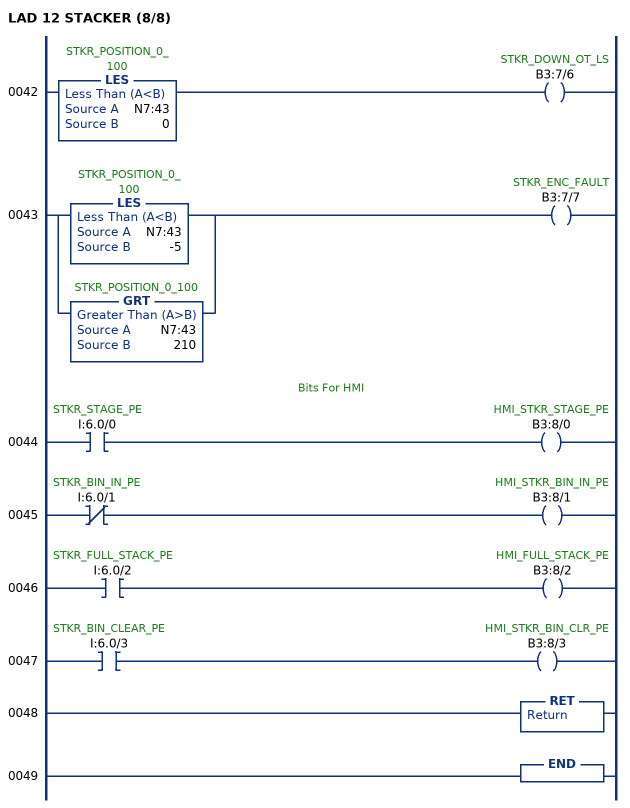
% Rung: 42 %
SOR LES N7:43 0 OTE B3:7/6 EOR
%   N7:43  STKR_POSITION_0_100 %
%   B3:7/6  STKR_DOWN_OT_LS %
% Rung: 43 %
SOR BST LES N7:43 -5 NXB GRT N7:43 210 BND OTE B3:7/7 EOR
%   N7:43  STKR_POSITION_0_100 %
%   B3:7/7  STKR_ENC_FAULT %
% Rung: 44 %
% Bits For HMI %
SOR XIC I:6.0/0 OTE B3:8/0 EOR
%   I:6.0/0  STKR_STAGE_PE %
%   B3:8/0  HMI_STKR_STAGE_PE %
% Rung: 45 %
SOR XIO I:6.0/1 OTE B3:8/1 EOR
%   I:6.0/1  STKR_BIN_IN_PE %
%   B3:8/1  HMI_STKR_BIN_IN_PE %
% Rung: 46 %
SOR XIC I:6.0/2 OTE B3:8/2 EOR
%   I:6.0/2  STKR_FULL_STACK_PE %
%   B3:8/2  HMI_FULL_STACK_PE %
% Rung: 47 %
SOR XIC I:6.0/3 OTE B3:8/3 EOR
%   I:6.0/3  STKR_BIN_CLEAR_PE %
%   B3:8/3  HMI_STKR_BIN_CLR_PE %
% Rung: 48 %
SOR RET EOR
% Rung: 49 %
SOR END EOR

OTHER DOCUMENTED ADDRESSES
  B3:0/9  SANITIZE_LTCH  "Triggered by reset limit sw."
  B3:0/10  SANITIZE_BIT  "Allow crdl ltch2 to unlatch only once until sanitize cycle is over"
  B3:0/11  CRDL_EN  "mcr on and no encoder fault"
  B3:0/15  CRDL_HAND_SS
  B3:1/1  RINSE_SELECT  "Turn ON Rinse"
  B3:1/9  RINSE_TEST
  B3:1/14  DUMP_INTERLOCK_SEL  "Dump Wash interlock"
  B3:2/7  UPPER_WASH_TEST
  B3:3/0  OPEN_CONTACT  "Machine not Equipt with OT LS"
  B3:3/9  FILTER_FLUSH_ON  "HMI Turn On Filter Flush"
  B3:3/11  MANUAL_BRUSH_DR_IN
  B3:3/12  MANUAL_BRUSH_DR_OUT
  B3:4/0  HMI_PID_MODE
  B3:4/1  HMI_PID_ALARM
  B3:6/11  BIN_STOP_DWN_SS
  C5:0/CU  EVENT_COUNTER
  F8:6  RAW_OUT_TO_VFD
  I:2.0/2  CHECK_MOTOR_OLS  "MP1,2,3,4,5"
  I:2.0/3  HP_PUMP_RUNNING
  I:2.0/4  CRADLE_VFD_RUNNING
  I:2.0/5  BRUSH_VFD_RUNNING
  I:2.0/6  XFER_PUMP_VFD_RUNNIN
  I:2.0/7  CRADLE_TORQUE_LIMIT
  I:5.0/3  BRUSH_GOING_IN
  I:5.0/4  BRUSH_GOING_OUT
  I:5.0/5  CRADLE_IN_MOTION
  I:5.0/6  BRUSH_RUNNING
  I:5.0/7  XFER_PUMP_RUNNING
  I:6.0  MAIN_TANK_RAW
  I:6.0/4  STKR_HI_LIMIT  "PROXIMITY SENSOR"
  L10:1/1  FAULT_MESSAGES
  N7:1/0  "Fault-Infeed Blocked"
  N7:1/1  "Fault-Outfeed Blocked"
  N7:1/2  "Fault-Cradle Overtravel Up"
  N7:1/3  "Fault-Cradle Overtravel down"
  N7:1/4  "Fault-Torque Cradle Inverter"
  N7:1/5  "Main Tank Low"
  N7:1/6  "Encoder Fault"
  N7:1/7  "Fill Main Tank"
  N7:10  FILTER_LOW_LS  "Filter Tank Low Level LS"
  N7:32  HP_PID_OUTPUT  "0-16383"
  N7:36  HMI_FLUSH_VALVE  "HMI TIME BETWEEN FLUSH"
  N7:37  HMI_FLUSH_VALVE_  "HMI FLUSHING TIME"
  N7:59  BIN_D_SLOW_DOWN
  N7:60  CATWALK_OPS_TIMER
  N9:0  K1
  O:0.0/7  CRADLE_COAST_TO_STOP  "MI2"
  O:0.0/12  FI
  O:0.1  OUT_TO_HP_VFD
  PD11:1  HIGH_PRESS_PUMP_PID
  PD11:1.2  PRESSURE_SP
  PD11:1.3  HP_KC
  PD11:1.4  HP_TI
  PD11:1.5  HP_TD
  PD11:1.13  LOOP_UPDATE_TIME  ".002"
  PD12:0.3  HP_PUMP_PID
  STKR_FULL_UP  
  T4:0/EN  CRDL_DWN_T  "Allows cradle to set down completely before conv starts"
  T4:1  CRDL_FLT_T1
  T4:2  CRDL_FLT_T2
  T4:5  CLEAN_CW_TMR  "CLOCKWISE CLEANING TIME"
  T4:6  SANITIZE_T
  T4:7  CRDL_DWN_T2  "Inhibits cradle up for 5 sec. after cradle sets down"
  T4:8  CLEAN_CCW  "COUNTER CLOCKWISE CLEANING TIME"
  T4:10  CRADLE_TIMER  "Cradle travel watch dog timer"
  T4:28/DN  LS_MED_BIN_DELAY
  T4:33/DN  STKR_RESTART_DELAY
  T4:34/DN  BIN_IN_DLY  "Stacker going down"
  T4:42  "stop delay 1234"

COMMENTS NOT ATTACHED TO A CURRENT RUNG
  N7:1/0: As long as the bit is set, the message will be displayed.  Bit #1 is Message #1.  Bit #3 is message #4.  Binary to decimal.
  T4:6.PRE: As long as the bit is set, the message will be displayed.  Bit #1 is Message #1.  Bit #3 is message #4.  Binary to decimal.
  T4:7: Timer not used

REVISION NOTES
  0: Added barrier and overtravel tatches
  1: Added indepentent barrier and overtravel catches
  2: Changed ffrom Panel #8.  Added B3:0/1 to prevent B3:0/5 from latching up while cradle is not down
  3: Added more troubleshooting help - step sequences
  4: Costa Rica Panel #19 with individual upper and lower wash solenoids

DATA TABLE (non-zero values as saved)
DATA B3
% B3:0 % 0X0DDA 0X5003 0X0770 0X0000 0X3D00 0X051C 0X001D 0X8402 0X0014 0X0000
DATA T4
% .PRE .ACC %
% T4:0 % 50 50
% T4:1 % 1 0
% T4:2 % 1 0
% T4:3 % 500 0
% T4:4 % 2 0
% T4:5 % 5 5
% T4:6 % 658 0
% T4:7 % 375 500
% T4:8 % 5 5
% T4:9 % 2 2
% T4:10 % 500 0
% T4:11 % 75 0
% T4:12 % 150 0
% T4:13 % 120 41
% T4:14 % 100 0
% T4:15 % 10 0
% T4:16 % 10 0
% T4:17 % 500 0
% T4:18 % 2 2
% T4:19 % 300 277
% T4:20 % 10 0
% T4:21 % 3 0
% T4:22 % 3 0
% T4:23 % 3 0
% T4:24 % 3 0
% T4:25 % 4 4
% T4:26 % 50 50
% T4:27 % 15 15
% T4:28 % 2 2
% T4:29 % 2 0
% T4:30 % 7 7
% T4:31 % 5 5
% T4:32 % 10 0
% T4:33 % 25 0
% T4:34 % 4 0
% T4:35 % 3 0
% T4:36 % 3 3
% T4:37 % 4 0
% T4:38 % 60 0
% T4:39 % 100 100
% T4:40 % 10 10
% T4:41 % 5 0
% T4:42 % 1 2
DATA N7
% N7:0 % 86 0 10 102 101 22 27 72 0 0
% N7:10 % 0 0 12122 1 1 0 2 70 11468 11795
% N7:20 % 72 0 0 49 100 5 1 0 2 0
% N7:30 % 0 -8179 0 4000 80 -175 0 0 3 25
% N7:40 % 4 5833 6822 83 67 100 80 117 70 56
% N7:50 % 89 28 108 65 9 8 8 8 9 0
% N7:60 % 0 4000
DATA F8
% F8:0 % 2106 4095 4046 12122 3
% F8:5 % 0 0 3 0 0
